// TwinCAT 3 PLC project Untitled1
// ProgramVersion: 3.1.4022.2
// libraries:
//   Tc2_Standard, * (Beckhoff Automation GmbH)
//   Tc2_System, * (Beckhoff Automation GmbH)
//   Tc3_EventLogger, * (Beckhoff Automation GmbH)
//   Tc3_Module, * (Beckhoff Automation GmbH)
// project tree:
//   / PlcTask.TcTTO (not stored)
//   POUs/ MAIN.TcPOU, ConfirmableAlarmWithArguments.TcPOU, AlarmWithCustomSourceInfo.TcPOU, SendMessage.TcPOU
// real-time tasks:
//   TASK PlcTask: cycle T#10ms, priority 20, ADS port 350

// ---- POUs/MAIN.TcPOU
PROGRAM MAIN

SendMessage();
ConfirmableAlarmWithArguments();
AlarmWithCustomSourceInfo();

END_PROGRAM

// ---- POUs/SendMessage.TcPOU
PROGRAM SendMessage
VAR
    bIsInitalized : BOOL;
    fbMessage : FB_TcMessage;
    bSendMessage : BOOL;
END_VAR

IF NOT bIsInitalized THEN
    bIsInitalized := TRUE;
    fbMessage.CreateEx(TC_Events.MyEvents.Start, 0);
END_IF

IF bSendMessage THEN
    bSendMessage := FALSE;
    fbMessage.Send(0);
END_IF

END_PROGRAM

// ---- POUs/ConfirmableAlarmWithArguments.TcPOU
PROGRAM ConfirmableAlarmWithArguments
VAR
    bIsInitalized : BOOL;
    
    fbAlarm : FB_TcAlarm;
    bRaiseAlarm : BOOL;
    bClearAlarm : BOOL;
    bConfirmAlarm : BOOL;
END_VAR

IF NOT bIsInitalized THEN
	bIsInitalized := TRUE;
	fbAlarm.CreateEx(TC_Events.MyEvents.Stop, TRUE, 0);	
END_IF

IF bRaiseAlarm THEN
	bRaiseAlarm := FALSE;
	fbAlarm.ipArguments.Clear().AddString('Alice');
	fbAlarm.Raise(0);
END_IF

IF bConfirmAlarm THEN
	bConfirmAlarm := FALSE;
	fbAlarm.Confirm(0);
END_IF

IF bClearAlarm THEN
	bClearAlarm := FALSE;
	fbAlarm.Clear(0, FALSE);
END_IF

END_PROGRAM

// ---- POUs/AlarmWithCustomSourceInfo.TcPOU
PROGRAM AlarmWithCustomSourceInfo
VAR
    bIsInitalized : BOOL;
    fbAlarm : FB_TcAlarm;
    bRaiseAlarm : BOOL;
    bClearAlarm : BOOL;
    fbSourceInfo : FB_TcSourceInfo;
END_VAR

IF NOT bIsInitalized THEN
    bIsInitalized := TRUE;
    fbSourceInfo.Clear();
    fbSourceInfo.sName := 'Water pump 3';
    fbAlarm.CreateEx(TC_Events.MyEvents.Stop, FALSE, fbSourceInfo);
END_IF

IF bRaiseAlarm THEN
    bRaiseAlarm := FALSE;
    fbAlarm.ipArguments.Clear().AddString('Bob');
    fbAlarm.Raise(0);
END_IF

IF bClearAlarm THEN
    bClearAlarm := FALSE;
    fbAlarm.Clear(0, TRUE);
END_IF

END_PROGRAM
